FUNCTION F_Generic_To_LREAL : LREAL
VAR_INPUT
	 Value : T_Generic;
END_VAR
VAR	
	pBool			: POINTER TO BOOL;
    pByte			: POINTER TO BYTE;
    pWord			: POINTER TO WORD;
    pDWord			: POINTER TO DWORD;
    pLWord			: POINTER TO LWORD;
    pSint			: POINTER TO SINT;
    pInt			: POINTER TO INT;
    pDint			: POINTER TO DINT;
    pLint			: POINTER TO LINT;
    pUSint			: POINTER TO USINT;
    pUInt			: POINTER TO UINT;
    pUDint			: POINTER TO UDINT;
    pULint			: POINTER TO ULINT;
    pReal			: POINTER TO REAL;
    pLReal			: POINTER TO LREAL;
    pString			: POINTER TO STRING(255);
    pWString		: POINTER TO WSTRING;
    pTime			: POINTER TO TIME;
    pDate			: POINTER TO DATE;
    pDate_And_Time	: POINTER TO DATE_AND_TIME;
    pTime_Of_Day	: POINTER TO TIME_OF_DAY;
    pPointer		: PVOID;
	pLTime 			: POINTER TO LTIME;
END_VAR

IF Value.pValue = 0 THEN RETURN; END_IF;

CASE Value.TypeClass OF 
	__SYSTEM.TYPE_CLASS.TYPE_BOOL:
		pBool := Value.pValue;
		F_Generic_To_LREAL := TO_LREAL(pBool^);
		
    __SYSTEM.TYPE_CLASS.TYPE_BYTE:
		pByte := Value.pValue;
		F_Generic_To_LREAL := TO_LREAL(pByte^);
		
    __SYSTEM.TYPE_CLASS.TYPE_WORD:
		pWord := Value.pValue;
		F_Generic_To_LREAL := TO_LREAL(pWord^);
		
    __SYSTEM.TYPE_CLASS.TYPE_DWORD:
		pDWord := Value.pValue;
		F_Generic_To_LREAL := TO_LREAL(pDWord^);
		
    __SYSTEM.TYPE_CLASS.TYPE_LWORD:
		pLWord := Value.pValue;
		F_Generic_To_LREAL := TO_LREAL(pLWord^);
		
    __SYSTEM.TYPE_CLASS.TYPE_SINT:
		pSint := Value.pValue;
		F_Generic_To_LREAL := TO_LREAL(pSint^);
		
    __SYSTEM.TYPE_CLASS.TYPE_INT:
		pInt := Value.pValue;
		F_Generic_To_LREAL := TO_LREAL(pInt^);
		
    __SYSTEM.TYPE_CLASS.TYPE_DINT:
		pDint := Value.pValue;
		F_Generic_To_LREAL := TO_LREAL(pDint^);
		
    __SYSTEM.TYPE_CLASS.TYPE_LINT:
		pLint := Value.pValue;
		F_Generic_To_LREAL := TO_LREAL(pLint^);
		
    __SYSTEM.TYPE_CLASS.TYPE_USINT:
		pUSint := Value.pValue;
		F_Generic_To_LREAL := TO_LREAL(pUSint^);
		
    __SYSTEM.TYPE_CLASS.TYPE_UINT:
		pUInt := Value.pValue;
		F_Generic_To_LREAL := TO_LREAL(pUInt^);
		
    __SYSTEM.TYPE_CLASS.TYPE_UDINT:
		pUDint := Value.pValue;
		F_Generic_To_LREAL := TO_LREAL(pUDint^);
		
    __SYSTEM.TYPE_CLASS.TYPE_ULINT:
		pULint := Value.pValue;
		F_Generic_To_LREAL := TO_LREAL(pULint^);
		
   __SYSTEM.TYPE_CLASS.TYPE_REAL:
		pReal := Value.pValue;
		F_Generic_To_LREAL := TO_LREAL(pReal^);
		
    __SYSTEM.TYPE_CLASS.TYPE_LREAL:
		pLReal := Value.pValue;
		F_Generic_To_LREAL := TO_LREAL(pLReal^);
		
    __SYSTEM.TYPE_CLASS.TYPE_STRING:
		pString := Value.pValue;
		F_Generic_To_LREAL := TO_LREAL(pString^);
		
   __SYSTEM.TYPE_CLASS.TYPE_WSTRING:
		pWString := Value.pValue;
		F_Generic_To_LREAL := TO_LREAL(pWString^);
		
    __SYSTEM.TYPE_CLASS.TYPE_TIME:
		pTime := Value.pValue;
		F_Generic_To_LREAL := TO_LREAL(pTime^);
		
    __SYSTEM.TYPE_CLASS.TYPE_DATE:
		pDate := Value.pValue;
		F_Generic_To_LREAL := TO_LREAL(pDate^);
		
    __SYSTEM.TYPE_CLASS.TYPE_DATEANDTIME:
		pDate_And_Time := Value.pValue;
		F_Generic_To_LREAL := TO_LREAL(pDate_And_Time^);
		
    __SYSTEM.TYPE_CLASS.TYPE_TIMEOFDAY:
		pTime_Of_Day := Value.pValue;
		F_Generic_To_LREAL := TO_LREAL(pTime_Of_Day^);
	
	__SYSTEM.TYPE_CLASS.TYPE_POINTER:
		F_Generic_To_LREAL := TO_LREAL(Value.pValue);
		
	__SYSTEM.TYPE_CLASS.TYPE_LTIME:
		pLTime := Value.pValue;
		F_Generic_To_LREAL := TO_LREAL(pLTime^);
END_CASE

END_FUNCTION

(* stored: Version 1.1.0.1, ProductVersion 3.1.4024.4
   POU F_Generic_To_LREAL: Id {8fc0ddb6-486d-4a36-bd95-15d4cb9dd2f7}, SpecialFunc None *)
